Fanuc KAREL source: kb00002.compact.KL

PROGRAM KB00002
%STACKSIZE=65535
%PRIORITY=65535
%NOLOCKGROUP
VAR
P1 : INTEGER
RESULT : INTEGER
BEGIN
P1=1
RESULT=ABS(P1)
END KB00002
